FUNCTION_BLOCK UnitTest
VAR_INPUT
END_VAR
VAR_OUTPUT
END_VAR
VAR
    _testSuite: ITestSuite;
END_VAR

METHOD FB_init : BOOL
VAR_INPUT
	bInitRetains : BOOL; // if TRUE, the retain variables are initialized (warm start / cold start)
	bInCopyCode : BOOL;  // if TRUE, the instance afterwards gets moved into the copy code (online change)
    _testSuite: ITestSuite;
END_VAR
THIS^._testSuite := _testSuite;
END_METHOD

PROPERTY testSuite : ITestSuite
GET
testSuite := THIS^._testSuite;
END_GET
SET
END_SET
END_PROPERTY

END_FUNCTION_BLOCK

(* stored: Version 1.1.0.1, ProductVersion 3.1.4022.12
   POU UnitTest: Id {ea4359ae-5c6a-467c-98f8-171e8d268a16}, SpecialFunc None
   Method FB_init: Id {6b3fd7b1-247d-4dbb-a886-62531fb1251a}
   Property testSuite: Id {db19b493-ce6b-492a-a438-736ac3fb3ae0}
   Get Get: Id {01b8d9d6-5b50-44e1-a44e-4b20f2c38f41}
   Set Set: Id {1281dcda-0757-4b75-94fd-4c5618ba9b5d} *)
